{library PUBLIC}
(* Level 1 function to write strobe value.
    Do not call this function from applications if functions on level 2-6 are used. *)
FUNCTION NodeWriteStrobe : BOOL
VAR_INPUT
	Address: 		INT;		(* Address, use the function ToAddress() to convert station and device number to a valid address. *)
	Value:			BOOL;		(* New strobe value. *)
END_VAR
VAR
	AWord:			WORD;
END_VAR

CASE NodeGetType(Address) OF
	DEVICE_TYPE.TYPE_ABB_1:  (* ABB Robot *)
		AWord:=ComGVL._qwABB;
		AWord.15:=Value;
		ComGVL._qwABB:=AWord;

	DEVICE_TYPE.TYPE_GANTRY_1:  (* Gantry robot *)
		AWord.15:=Value;
		(* Empty no real strobe *)


	DEVICE_TYPE.TYPE_SIMULATED:
		ComGVL._DataSimulatedStation[1, 1]:=BOOL_TO_BYTE(Value);
		AWord.15:=Value;
ELSE
		AWord:=0;
		AWord.15:=Value;
END_CASE;

(* Return value *)
NodeWriteStrobe:=AWord.15;

END_FUNCTION

(* stored: Version 1.1.0.1, ProductVersion 3.1.4024.2
   POU NodeWriteStrobe: Id {0822df44-2beb-4972-994c-53aff074438b}, SpecialFunc None *)
